{attribute 'qualified_only'}
{attribute 'strict'}
TYPE E_HMI_TIP_TILT_TABS :
(
	TIP_A,
    TIP_B,
	TILT_A,
    TILT_B

);
END_TYPE

(* stored: Version 1.1.0.1, ProductVersion 3.1.4024.14
   DUT E_HMI_TIP_TILT_TABS: Id {f5f104c4-76d5-4352-802e-f58bb69541e3} *)
